// TwinCAT 3 PLC project WasherController
// ProgramVersion: 3.1.4024.0
// libraries:
//   Tc2_Standard, * (Beckhoff Automation GmbH)
//   Tc2_System, * (Beckhoff Automation GmbH)
//   Tc3_Module, * (Beckhoff Automation GmbH)
//   VisuSymbols,3.5.10.0,System
// project tree:
//   / GlobalTextList.TcGTLO, PlcTask.TcTTO, 视图管理器.TcVMO (not stored)
//   POUs/ MAIN.TcPOU, ServoControl.TcPOU, Spray.TcPOU
//   VISUs/ Visualization.TcVIS
// real-time tasks:
//   TASK PlcTask: cycle T#10ms, priority 20, ADS port 350

CONFIGURATION WasherController
    RESOURCE PLC ON TwinCAT3
        TASK PlcTask(INTERVAL := T#10ms, PRIORITY := 20);
        PROGRAM MAIN WITH PlcTask : MAIN;
    END_RESOURCE
END_CONFIGURATION

// ---- POUs/MAIN.TcPOU
PROGRAM MAIN
VAR
	ServoDo:BOOL;
	ServoDone: BOOL;
	ServoAngle:REAL;
	CurrentAngle:REAL;
	FixtureEnable:BOOL;
	Controller:ServoControl;
	//Spray block
	spray:Spray;
	SprayExecute:BOOL:=TRUE;
	
	Order:ARRAY[0..7] OF INT:=[1,2,3,4,5,6,7,8];
	//get spin before servo step to get 1 at head
	FixtureState:INT:=0;
	temp:INT:=0;
	FixtureStateArray:ARRAY[0..7] OF BOOL:=[0,0,0,0,0,0,0,0];
	i: INT;
END_VAR

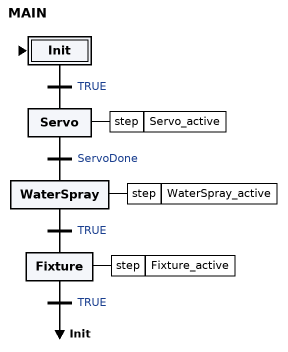
INITIAL_STEP Init:
END_STEP
TRANSITION FROM Init TO Servo
    := TRUE;
END_TRANSITION
STEP Servo:
    Servo_active(N);  // step action
END_STEP
TRANSITION FROM Servo TO WaterSpray
    := ServoDone;
END_TRANSITION
STEP WaterSpray:
    WaterSpray_active(N);  // step action
END_STEP
TRANSITION FROM WaterSpray TO Fixture
    := TRUE;
END_TRANSITION
STEP Fixture:
    Fixture_active(N);  // step action
END_STEP
TRANSITION FROM Fixture TO Init
    := TRUE;
END_TRANSITION

ACTION Fixture_active:
temp:=1;
FOR i:=0 TO 7 DO
	FixtureStateArray[i]:= INT_TO_BOOL(REAL_TO_INT(FixtureState/temp) MOD 2);
	temp:=temp*2;
END_FOR
END_ACTION

ACTION Servo_active:
Controller(
	bExecute:=ServoDo,
	bDone=>ServoDone,
	Order=>Order,
	CurrentAngle=>CurrentAngle
);
END_ACTION

ACTION WaterSpray_active:
spray(bExecute:=SprayExecute,
	Order:=Order,
	Angle:=CurrentAngle,
	bDone=>
);
END_ACTION

END_PROGRAM

// ---- POUs/ServoControl.TcPOU
FUNCTION_BLOCK ServoControl
VAR_INPUT
	bExecute:BOOL;
END_VAR
VAR_OUTPUT
	bDone:BOOL:=FALSE;
	Order:ARRAY[0..7] OF INT:=[2,3,4,5,6,7,8,1];
	CurrentAngle:REAL;
END_VAR
VAR
	ServoBlock:BOOL:=FALSE;
	MoveStart:BOOL:=FALSE;
	MoveFinish:BOOL:=TRUE;
	initAngle:REAL:=0;
	Step:REAL:=-45;
	AnglePush:REAL;
	
	//StatePull:BOOL:=FALSE;
	Angles:ARRAY[0..7] OF REAL:=[0.0,0.0,0.0,0.0,90.0,180.0,180.0,90.0];
	temp:REAL;
	temp_order:INT;
	//该模块第一次运行为到达原点
END_VAR

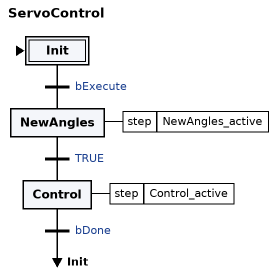
INITIAL_STEP Init:
END_STEP
TRANSITION FROM Init TO NewAngles
    := bExecute;
END_TRANSITION
STEP NewAngles:
    NewAngles_active(N);  // step action
END_STEP
TRANSITION FROM NewAngles TO Control
    := TRUE;
END_TRANSITION
STEP Control:
    Control_active(N);  // step action
END_STEP
TRANSITION FROM Control TO Init
    := bDone;
END_TRANSITION

ACTION Control_active:
IF NOT ServoBlock THEN
	
	//StatePull:=FALSE;
	MoveStart:=TRUE;
	bDone:=MoveFinish;
	IF bDone = TRUE THEN
		MoveStart:=FALSE;
		IF initAngle < -359 THEN
			initAngle:= 0;
		END_IF
		initAngle:=initAngle+Step;
		MoveFinish:=FALSE;
	END_IF
END_IF
END_ACTION

ACTION NewAngles_active:
IF NOT ServoBlock THEN
	temp:=Angles[0];
	Angles[0]:=Angles[1];
	Angles[1]:=Angles[2];
	Angles[2]:=Angles[3];
	Angles[3]:=Angles[4];
	Angles[4]:=Angles[5];
	Angles[5]:=Angles[6];
	Angles[6]:=Angles[7];
	Angles[7]:=temp;
	//Order in world frame
	temp_order:=Order[7];
	Order[7]:=Order[6];
	Order[6]:=Order[5];
	Order[5]:=Order[4];
	Order[4]:=Order[3];
	Order[3]:=Order[2];
	Order[2]:=Order[1];
	Order[1]:=Order[0];
	Order[0]:=temp_order;
	
	AnglePush:=initAngle;
	bDone:=FALSE;
END_IF
END_ACTION

END_FUNCTION_BLOCK

// ---- POUs/Spray.TcPOU
FUNCTION_BLOCK Spray
VAR_INPUT
	bExecute:BOOL;
	Order:ARRAY[0..7] OF INT;//世界坐标系下的夹具次序
	Angle:REAL;
END_VAR
VAR_OUTPUT
	bDone: BOOL;
END_VAR
VAR
	pick:INT;
	SpraySwitch:ARRAY[0..7] OF BOOL:=[0,0,0,0,0,0,0,0];//Order by Eletronic
	SwitchOpen:ARRAY[0..7] OF INT:=[0,0,0,0,0,0,0,0];//Order by Eletronic
	Angle2Switch:ARRAY[0..7] OF INT:=[3,2,1,8,7,6,5,4];
	SensorSignal:BOOL:=TRUE;
	i: INT;
END_VAR

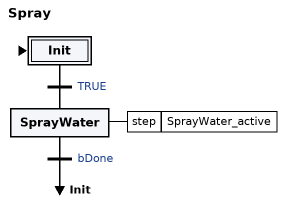
INITIAL_STEP Init:
END_STEP
TRANSITION FROM Init TO SprayWater
    := TRUE;
END_TRANSITION
STEP SprayWater:
    SprayWater_active(N);  // step action
END_STEP
TRANSITION FROM SprayWater TO Init
    := bDone;
END_TRANSITION

ACTION SprayWater_active:
pick:= REAL_TO_INT(Angle/(-45));
IF pick = 8 THEN
	pick:=0;
END_IF
IF SensorSignal THEN
	//By Order
	//SpraySwitch[Order[2]-1]:=TRUE;
	//SwitchOpen[Order[2]-1]:=SwitchOpen[Order[2]-1]+1;
	//By Angle
	SpraySwitch[Angle2Switch[pick]-1]:=TRUE;
	SwitchOpen[Angle2Switch[pick]-1]:=SwitchOpen[Angle2Switch[pick]-1]+1;
END_IF
SensorSignal:=FALSE;
//SpraySwitch[Order[3]-1]:=FALSE;

IF pick=0 THEN
	SpraySwitch[Angle2Switch[7]-1]:=FALSE;
	SwitchOpen[Angle2Switch[7]-1]:=0;
ELSE
	SpraySwitch[Angle2Switch[pick-1]-1]:=FALSE;
	SwitchOpen[Angle2Switch[pick-1]-1]:=0;
END_IF

FOR i := 0 TO 7 DO
	IF SwitchOpen[i]>=20 THEN
		SpraySwitch[i]:=FALSE;
		SwitchOpen[i]:=0;
	END_IF
END_FOR
END_ACTION

END_FUNCTION_BLOCK

// ---- GlobalTextList.TcGTLO
TEXTLIST GlobalTextList
  708 = '%.2f'
  508 = '%d'
  831 = 'No1 夹具位置：%d'
  612 = '喷水'
  850 = '喷水阀门'
  510 = '夹具'
  989 = '电机'
  688 = '电机启动'
  223 = '角度：%.2f'
END_TEXTLIST

// ---- VISUs/Visualization.TcVIS
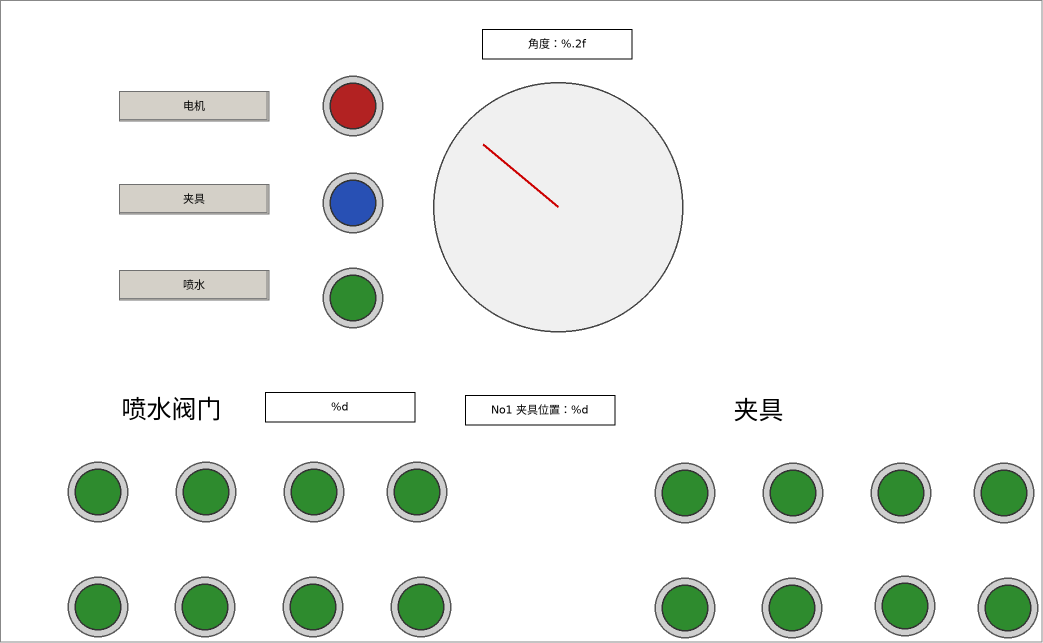
VISUALIZATION Visualization  // 1043x643
    Button (119,91 150x30), "电机"
        OnMouseClick: execute { MAIN.ServoDo :=NOT MAIN.ServoDo; }
    Meter360 (433,82 250x250), value: MAIN.Controller.CurrentAngle, style: Meter-Meter360-Red, scale format: %.1f, scale 0..360
    Button (119,270 150x30), "喷水"
        OnMouseClick: execute { MAIN.SprayExecute:= NOT MAIN.SprayExecute; }
    Button (119,184 150x30), "夹具"
        OnMouseClick: execute { MAIN.FixtureEnable:= NOT MAIN.FixtureEnable; }
    Lamp1 (318,71 70x70), variable: MAIN.ServoDo, style: Lamp-Lamp1-Red
    Lamp1 (318,168 70x70), variable: MAIN.FixtureEnable, style: Lamp-Lamp1-Blue
    Lamp1 (318,263 70x70), variable: MAIN.SprayExecute, style: Lamp-Lamp1-Green
    Lamp1 (63,457 70x70), variable: MAIN.spray.SpraySwitch[0], style: Lamp-Lamp1-Green
    Lamp1 (171,457 70x70), variable: MAIN.spray.SpraySwitch[1], style: Lamp-Lamp1-Green
    Lamp1 (279,457 70x70), variable: MAIN.spray.SpraySwitch[2], style: Lamp-Lamp1-Green
    Lamp1 (382,457 70x70), variable: MAIN.spray.SpraySwitch[3], style: Lamp-Lamp1-Green
    Lamp1 (63,572 70x70), variable: MAIN.spray.SpraySwitch[4], style: Lamp-Lamp1-Green
    Lamp1 (170,572 70x70), variable: MAIN.spray.SpraySwitch[5], style: Lamp-Lamp1-Green
    Lamp1 (278,572 70x70), variable: MAIN.spray.SpraySwitch[6], style: Lamp-Lamp1-Green
    Lamp1 (386,572 70x70), variable: MAIN.spray.SpraySwitch[7], style: Lamp-Lamp1-Green
    Label (65,390 213x38), "喷水阀门"
    Rectangle (482,29 150x30), "角度：%.2f", text variable: MAIN.Controller.CurrentAngle
    Rectangle (265,392 150x30), "%d", text variable: MAIN.spray.Order[2]
    Rectangle (465,395 150x30), "No1 夹具位置：%d", text variable: MAIN.spray.pick+1
    Lamp1 (650,458 70x70), variable: MAIN.FixtureStateArray[0], style: Lamp-Lamp1-Green
    Lamp1 (758,458 70x70), variable: MAIN.FixtureStateArray[1], style: Lamp-Lamp1-Green
    Lamp1 (866,458 70x70), variable: MAIN.FixtureStateArray[2], style: Lamp-Lamp1-Green
    Lamp1 (969,458 70x70), variable: MAIN.FixtureStateArray[3], style: Lamp-Lamp1-Green
    Lamp1 (650,573 70x70), variable: MAIN.FixtureStateArray[4], style: Lamp-Lamp1-Green
    Lamp1 (757,573 70x70), variable: MAIN.FixtureStateArray[5], style: Lamp-Lamp1-Green
    Lamp1 (870,571 70x70), variable: MAIN.FixtureStateArray[6], style: Lamp-Lamp1-Green
    Lamp1 (973,573 70x70), variable: MAIN.FixtureStateArray[7], style: Lamp-Lamp1-Green
    Label (652,391 213x38), "夹具"
END_VISUALIZATION
